# B&R Automation Studio project warcabot
Automation Studio 6.7.0.187; technology packages: mappMotion 6.7.2, mappView 6.7.0, OpcUaCs 6.7.0

## Configuration Config1

### Task classes (Cpu.sw)
```
Cyclic#4:
  TestOpcua <- TestOpcua.prg
Libraries: McBase, MpBase
```

### Hardware
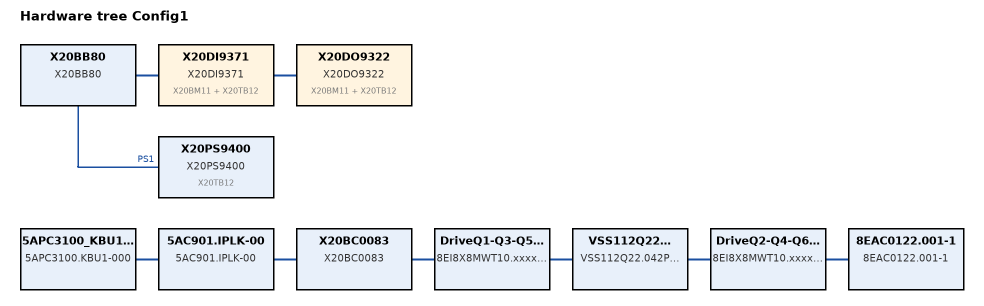
```
5AC901.IPLK-00 : 5AC901.IPLK-00 v2.1.0.0  [SL -> 5APC3100_KBU1_000.SL2]
5APC3100_KBU1_000 : 5APC3100.KBU1-000 v2.3.1.0
  Connector IF3:
    AssignedOperatingSystem = ARemb
    ActivateDevice = 1
  Connector IF4:
    AssignedOperatingSystem = ARemb
    ActivateDevice = 1
  Connector IF5:
    AssignedOperatingSystem = ARemb
  Connector IF6:
    AssignedOperatingSystem = ARemb
  Connector IF7:
    AssignedOperatingSystem = ARemb
  Connector IF8:
    AssignedOperatingSystem = ARemb
  ConfigurationID = warcabot_Config1
  Simulation = 1
  FileDevice1
  FileDeviceName1 = USER
  FileDevicePath1 = USER_PATH
8EAC0122.001-1 : 8EAC0122.001-1 v3.0.0.0  [SS -> DriveQ2-Q4-Q6_Racer3_1.SS1]
DriveQ1-Q3-Q5_Racer3_1 : 8EI8X8MWT10.xxxx-1 v2.4.0.0 (NodeNumber=2)  [PLK1 -> X20BC0083.PLK2 [Cable Type=PowerlinkCable, Length=10, Version=1.0.0.3]; PLK2 -> VSS112Q22.042P-000.PLK1 [Cable Type=PowerlinkCable, Length=10, Version=1.0.0.3]]
DriveQ2-Q4-Q6_Racer3_1 : 8EI8X8MWT10.xxxx-1 v2.4.0.0 (NodeNumber=4)  [PLK1 -> VSS112Q22.042P-000.PLK2 [Cable Type=PowerlinkCable, Length=10, Version=1.0.0.3]]
VSS112Q22.042P-000 : VSS112Q22.042P-000 v1.11.0.929 (NodeNumber=3)  [PLK1 -> DriveQ1-Q3-Q5_Racer3_1.PLK2 [Cable Type=PowerlinkCable, Length=10, Version=1.0.0.3]; PLK2 -> DriveQ2-Q4-Q6_Racer3_1.PLK1 [Cable Type=PowerlinkCable, Length=10, Version=1.0.0.3]]
X20BB80 : X20BB80 v1.1.0.0
X20BC0083 : X20BC0083 v2.17.0.0 (NodeNumber=1)  [PLK1 -> 5AC901.IPLK-00.IF1 [Cable Type=PowerlinkCable, Length=10, Version=1.0.0.3]; PLK2 -> DriveQ1-Q3-Q5_Racer3_1.PLK1 [Cable Type=PowerlinkCable, Length=10, Version=1.0.0.3]; SL -> X20BB80.SL1]
X20BM11 : X20BM11 v1.1.0.0  [X2X1 -> X20BB80.IF1]
X20BM11_a : X20BM11 v1.1.0.0  [X2X1 -> X20BM11.X2X2]
X20DI9371 : X20DI9371 v1.6.1.0  [SS1 -> X20TB12.SS; SL -> X20BM11.SL1]
X20DO9322 : X20DO9322 v1.7.0.0  [SS1 -> X20TB12_b.SS; SL -> X20BM11_a.SL1]
X20PS9400 : X20PS9400 v1.9.0.0  [SS1 -> X20TB12_a.SS; PS -> X20BB80.PS1]
X20TB12 : X20TB12 v1.0.0.0
X20TB12_a : X20TB12 v1.0.0.0
X20TB12_b : X20TB12 v1.0.0.0
```

### Config.mpuserx - 5APC3100_KBU1_000/mappServices/Config.mpuserx
```
Element UserMgmtX (Type=mpuserx)
  mapp.Gen:
    Audit = TRUE
  UserMgmtSystem:
    UserMgmtSystemType = 0
  ServerSettings:
    Server = ADServer
      Timeout = 10
      Mapping:
        TableName
      DisplayName = username
      AdditionalUserData:
        [0] = mail
        [1] = telephoneNumber
  PasswordPolicy:
    PasswordMaxAge = 0
    PasswordExpirationNotification = 0
    PasswordHistory = 0
    PasswordChangeReq = FALSE
    PasswordCase = FALSE
    PasswordAlpha = FALSE
    PasswordSpecial = FALSE
    PasswordLength = 1
  UserAccount:
    InvalidPasswordAttempts = 3
    UserExpirationTime = 0
    AutoLogoutTime = 3600
    UserNameLength = 1
    NoDelete = FALSE
    AdminUnlockTime = 3600
    EditSameLevel = 1
  ImportExport:
    ImportUser = 2
    ImportRole = 2
    ImportUnchecked = FALSE
    FileChecksum = 2
  Users:
    DefUser#1:
      id = Admin
      name
      lang
      measSystem = 0
    DefUser#2:
      id = Oper
      name = Operator
      lang
      measSystem = 0
  Roles:
    DefRole#1:
      id = BR_SecurityAdmin
      level = 100
      admin = TRUE
    DefRole#2:
      id = Administrator
      level = 100
      admin = TRUE
    DefRole#3:
      id = Operator
      level = 20
      admin = FALSE
```

## Logical view

### Global.typ - Global data types
```iecst
TYPE
	PlayerColorEnum :
		(
		WHITE,
		BLACK
		);
	DifficultyLevelEnum :
		(
		HARD,
		MEDIUM,
		EASY
		);
	GameStateEnum :
		(
		WAITING_PLAYER, (*oczekiwanie na ruch gracza*)
		IDLE, (*oczekiwanie na rozpoczêcie gry*)
		CHECKING_MOVE, (*sprawdzanie poprawnoœci ruchu*)
		CHECKING_BOARD, (*weryfikacja planszy po ruchu*)
		ROBOT_MOVE, (*robot wykonuje ruch*)
		FINISHED (*koniec gry*)
		);
	PieceTypeEnum :
		(
		EMPTY,
		BLACK_KING,
		BLACK,
		WHITE_KING,
		WHITE
		);
	WinnerEnum :
		(
		ROBOT,
		PLAYER,
		NONE
		);
	PositionStruct : 	STRUCT
		Z : REAL;
		Y : REAL;
		X : REAL;
	END_STRUCT;
	MoveStruct : 	STRUCT
		TO_COLUMN : INT;
		TO_ROW : INT;
		FROM_COLUMN : INT;
		FROM_ROW : INT;
	END_STRUCT;
END_TYPE
```

### Global.var - Global variables
```iecst
VAR
	gTest : BOOL;
END_VAR
```

### Package Logical/Libraries - Global libraries

- Visualisation Logical/mappView (not shown)

### Program Logical/ManualCtrl

#### Variables.var
```iecst
VAR
	gRobotJog    : MpGroupJog;
	gRobotJogPar : MpGroupJogParType;
END_VAR

VAR CONSTANT

END_VAR
```

#### Cyclic.st
```iecst
PROGRAM _CYCLIC
	gRobotJog.MpLink := ADR(gAxesGroup);
	gRobotJog.Parameters := ADR(gRobotJogPar);
	gRobotJog.Enable := TRUE;

	gRobotJog();

END_PROGRAM
```

### Program Logical/Motion/Program

#### Main.st
```iecst
PROGRAM _INIT
	(* Insert code here *)
	gAxesGroup_Racer3_1;
	gAxisQ1_Racer3_1;
	gAxisQ2_Racer3_1;
	gAxisQ3_Racer3_1;
	gAxisQ4_Racer3_1;
	gAxisQ5_Racer3_1;
	gAxisQ6_Racer3_1;

END_PROGRAM

PROGRAM _CYCLIC
	(* Insert code here *)

END_PROGRAM

PROGRAM _EXIT
	(* Insert code here *)

END_PROGRAM
```

### Program Logical/TestOpcua

#### Main.st
```iecst
PROGRAM _INIT

	FOR i := 0 TO 63 DO
		gBoard[i] := 0;
	END_FOR;
	gBoard[0] := 1;
	gBoard[2] := 1;
	gBoard[4] := 1;
	gBoard[6] := 1;

	gBoard[9] := 1;
	gBoard[11] := 1;
	gBoard[13] := 1;
	gBoard[15] := 1;

	gBoard[16] := 1;
	gBoard[18] := 1;
	gBoard[20] := 1;
	gBoard[22] := 1;

	gBoard[41] := 2;
	gBoard[43] := 2;
	gBoard[45] := 2;
	gBoard[47] := 2;

	gBoard[48] := 2;
	gBoard[50] := 2;
	gBoard[52] := 2;
	gBoard[54] := 2;

	gBoard[57] := 2;
	gBoard[59] := 2;
	gBoard[61] := 2;
	gBoard[63] := 2;
	gGraStart := FALSE;
	gJakiKolor := FALSE;
	gCzyjaTura := FALSE;

END_PROGRAM

PROGRAM _CYCLIC
	(* Insert code here *)
	gTest;
END_PROGRAM

PROGRAM _EXIT
	(* Insert code here *)

END_PROGRAM
```
